# B&R Automation Studio project pneutrunk_plc (part 4)

#### pneutr2_reg_FF_stiff_data.c
```c
/*
 * pneutr2_reg_FF_stiff_data.c
 *
 * Academic License - for use in teaching, academic research, and meeting
 * course requirements at degree granting institutions only.  Not for
 * government, commercial, or other organizational use.
 *
 * Code generation for model "pneutr2_reg_FF_stiff".
 *
 * Model version              : 4.30
 * Simulink Coder version : 9.9 (R2023a) 19-Nov-2022
 * C source code generated on : Thu Feb 15 10:44:02 2024
 *
 * Target selection: bur_grt.tlc
 * Note: GRT includes extra infrastructure and instrumentation for prototyping
 * Embedded hardware selection: Intel->x86/Pentium
 * Code generation objectives: Unspecified
 * Validation result: Not run
 */

#include "pneutr2_reg_FF_stiff.h"

/* Constant parameters (default storage) */
const ConstP_pneutr2_reg_FF_stiff_T pneutr2_reg_FF_stiff_ConstP = {
  /* Expression: coef_1blue_1
   * Referenced by: '<Root>/Constant'
   */
  { 8.5717463150365491E-5, -1.5178110935199764E-6, -5.1507533201889129E-6,
    -4.0104560028142805E-7, -1.7129289185435491E-7, -4.4592625230545557E-7,
    -0.0024294858487422821, 3.9820571035780173E-5, 0.00014194348913824982,
    1.0779763981053751E-5, 4.8691806145412491E-6, 1.2240687126729779E-5,
    0.027186032468499655, -0.000390604161196484, -0.0015838551030587162,
    -0.00011698204244076088, -5.2523210718500108E-5, -0.00013650518202891186,
    -0.15170965057623756, 0.0017650946579940159, 0.0091350333868915647,
    0.00065126150638811556, 0.00027180379442720342, 0.000785516674273971,
    0.43233120736620573, -0.0034156500044472521, -0.028897920231378927,
    -0.0019455068426407257, -0.000689010003804365, -0.0024506052032467382,
    -0.54551465196653193, 0.0011895886985182566, 0.04928011865673651,
    0.002942446648700804, 0.0007337993722779018, 0.0040060166051372123,
    0.50512977080755284, -0.0047809288297403895, -0.03852433507794821,
    -0.0019253109483168883, -0.00010621822149096354, -0.0032474983289435574,
    0.2943360100687234, -0.0340414299034502, 0.038688128292281909,
    0.00078966690125624418, -0.0011243932202755762, 0.0011672777941613569 },

  /* Expression: coef_2green_1
   * Referenced by: '<Root>/Constant1'
   */
  { 3.5806457470463992E-5, 4.2068425285366185E-6, -2.307008943003239E-7,
    -2.8130907926246906E-7, 5.788444538503013E-7, -2.4818480944264519E-7,
    -0.0010926398714506292, -0.00010269300409286399, 5.9242568564171268E-6,
    7.716656677865785E-6, -1.4601073471851697E-5, 7.2919598185173952E-6,
    0.013304512173293481, 0.00098519204569556232, -7.8153808987968122E-5,
    -8.6901728962855031E-5, 0.00014548727107240185, -8.7693471415853716E-5,
    -0.082362007567461509, -0.0047066674356880328, 0.00060563468397506243,
    0.00051035549177713539, -0.00072968678478258365, 0.00055150404791877189,
    0.2700466009571485, 0.01163973248303852, -0.0025271867329235624,
    -0.0016371606003118366, 0.0019364089644989316, -0.0019042555969799237,
    -0.43174345718640667, -0.013838783021252042, 0.0052541678910867822,
    0.0027338218415489421, -0.0025985505984174404, 0.0034092802459716508,
    0.552385933579235, 0.0066940622681189946, -0.013604069710649497,
    -0.0020700479747369879, 0.0015023574386652, -0.0026069405140951157,
    0.031374405216318131, 0.00048138420611595288, -0.035622417341977054,
    0.00018286604488092231, -0.00022698979966827995, 0.0012027861166743492 },

  /* Expression: coef_2green_4
   * Referenced by: '<Root>/Constant10'
   */
  { 3.415320573463566E-7, 9.3053337461778723E-8, -1.1840409221532752E-7,
    -8.3671504125970439E-9, 3.5026579994580658E-9, -2.0473493718581922E-8,
    -2.0177539775413165E-5, -4.5777744650225739E-6, 5.1319620699227294E-6,
    4.6216124370471893E-7, -1.1677319901234268E-7, 9.3377979582771185E-7,
    0.00041167609423549265, 9.3021114154861822E-5, -9.1517441203400879E-5,
    -1.0160859722685084E-5, 1.4151670403326086E-6, -1.7147070588351255E-5,
    -0.0036565061339228488, -0.00098633859891033974, 0.000845215868210654,
    0.00011217230418689672, -6.5999698903405726E-6, 0.00016146662485588915,
    0.012721834814625485, 0.0057771156380495613, -0.0041345518318866188,
    -0.0006595704121746726, -4.6996251846852646E-6, -0.00082145775844466693,
    0.002615152654760115, -0.018645640174938138, 0.010129187197222871,
    0.0020683196398549757, 0.00014406107821792274, 0.0021836634425048385,
    0.20910235409508418, 0.032347602609962139, -0.022366862791594815,
    -0.0034592418366138264, -0.00038747013057998107, -0.0027517673928555875,
    -0.083971676633054743, -0.021473606225994771, -0.045616157291447669,
    0.0022934839006601539, 0.00025030061299072753, 0.0023621895615410903 },

  /* Expression: coef_2green_5
   * Referenced by: '<Root>/Constant11'
   */
  { 1.409263146447497E-6, -6.3007282692451016E-8, 1.1334083156168342E-8,
    9.230072254275008E-9, 2.74393730750942E-9, -4.8715649028139032E-8,
    -6.9391321709493125E-5, 2.0937049836852873E-6, -6.23736765151863E-7,
    -2.3185063573156576E-7, -5.5045992465423964E-8, 2.052665868062509E-6,
    0.0013210734825910666, -2.1292894715980217E-5, 8.565244556977659E-6,
    4.7322333858128524E-7, -1.1535975466056446E-7, -3.453185633002057E-5,
    -0.012145916271257683, 1.5971479419808272E-5, -2.3584719796187389E-5,
    3.192578938792718E-5, 9.9053898987882459E-6, 0.00029591296770094293,
    0.054487936398149417, 0.00099258756801452936, -0.00010064404267846677,
    -0.000347539885728757, -8.7991688376231036E-5, -0.0013616763907182364,
    -0.10407852174157033, -0.0062360441969368831, -0.00016216594324408893,
    0.0014800735016823512, 0.00033604108201676412, 0.0032439882128459277,
    0.3747821795642276, 0.015025591198706953, -0.0083042810415812855,
    -0.0030134939009767536, -0.00064323011865612925, -0.0036482215628668778,
    -0.004527716804257619, -0.010721196323413579, -0.065428003610548333,
    0.0021176098163992788, 0.00057191087607426664, 0.0025894065846387092 },

  /* Pooled Parameter (Expression: coef_2green_6)
   * Referenced by:
   *   '<Root>/Constant12'
   *   '<Root>/Constant18'
   */
  { 1.5081258956513881E-6, -9.046346810421332E-8, 1.4774610225232294E-7,
    -1.7432201593417331E-8, -2.0415701254911555E-9, -5.4201527217183439E-8,
    -7.3850872884215273E-5, 4.5089735689383433E-6, -6.9216959803445692E-6,
    9.8854099646194021E-7, 5.5053432274398986E-8, 2.2269085287207753E-6,
    0.0014042956430304265, -8.8061719814155312E-5, 0.00012698257113709691,
    -2.1915549658526132E-5, 9.0696936183742649E-8, -3.6440744397947455E-5,
    -0.012945155421301551, 0.00086167153240620023, -0.0011917294683145272,
    0.00024280347096503, -1.5415826108399811E-5, 0.00030134255124641181,
    0.058340999413557769, -0.0044888394554316634, 0.0063812751182880829,
    -0.0014299950795206462, 0.00018114458962297672, -0.0013129857525858957,
    -0.1100216315325513, 0.012310894186012916, -0.020155506459850911,
    0.0044334939497109281, -0.00089428426947732876, 0.0028179085747864164,
    0.3631415623276481, -0.01702695159348681, 0.021985457194170679,
    -0.0068753620174089982, 0.0020298400260213797, -0.0023791127843658631,
    0.075563804424678138, 0.010748302896753867, -0.0836195604466876,
    0.0040496210649481768, -0.0015285175321659943, 0.0017237408611272247 },

  /* Expression: coef_3yellow_2
   * Referenced by: '<Root>/Constant13'
   */
  { 6.4204697466336988E-5, -9.4342813666632677E-7, -3.98434162214021E-6,
    -2.4148886551485478E-7, 8.8600986529608742E-8, -3.529598140424027E-7,
    -0.0018407313544118249, 3.0510655304270148E-5, 0.00011104653151774753,
    6.5304832782381205E-6, -2.3344707108276623E-6, 9.65189940926156E-6,
    0.02097491538357809, -0.000387051166283223, -0.0012516712095343016,
    -7.179814137945989E-5, 2.3929248384559622E-5, -0.00010623259914238595,
    -0.12040940291919788, 0.0024820271108887929, 0.0072572354123937189,
    0.00040935377395097877, -0.00011913321761664191, 0.00059895110912360915,
    0.35915882237005048, -0.00861416236255178, -0.022717316237366777,
    -0.0012669750174637902, 0.00029353210289014188, -0.0018144810086714097,
    -0.49859157313593883, 0.015389607153086968, 0.036324219531468319,
    0.0020005131476629814, -0.0003405260446271574, 0.0028020994854614529,
    0.54244105552147959, -0.0045093597732031561, -0.020952154469339943,
    -0.0013450196814645764, 0.00026257246310186223, -0.0019162105937383018,
    0.29795717865338078, 0.029061424095047042, 0.019318582185105713,
    0.00054717765450625067, 0.00043700242127395092, 0.00039781477781437066 },

  /* Expression: coef_3yellow_3
   * Referenced by: '<Root>/Constant14'
   */
  { 6.48259537993542E-8, -1.7774373759257409E-7, -7.808320155327938E-8,
    3.8287288945787542E-8, 5.5727806872203979E-8, -1.8725128684800113E-8,
    -4.45539021636487E-6, 7.0819017739852445E-6, 3.6184317358179945E-6,
    -1.491338534879082E-6, -2.5306282351536662E-6, 8.3322003698335979E-7,
    0.0001039787062549207, -0.00011035727260183309, -6.5873046934394221E-5,
    2.2048281812537434E-5, 4.55402340551219E-5, -1.5071031926050898E-5,
    -0.00098793769743092826, 0.0008614769663412399, 0.00060282012366024156,
    -0.00015092450729609631, -0.00041124074118570862, 0.00014117705330117704,
    0.0022439189860935078, -0.0036459718424953552, -0.0030283199162596912,
    0.00044146382598600064, 0.001946472495698699, -0.00072655371363900109,
    0.018638716969889575, 0.0083590464791400559, 0.0087513807479669085,
    -0.00015550941198203396, -0.0045870757397633247, 0.0020466684533415095,
    0.22372555046354425, 0.00063339384125198669, -0.010561842394564404,
    -0.001534857218792919, 0.0046426063227622064, -0.0031765426227927333,
    0.21321109612687739, 0.062318293620291086, 0.0451142945040786,
    0.0030086997391691591, 0.00020377818613637877, 0.0025250451699678524 },

  /* Expression: coef_3yellow_4
   * Referenced by: '<Root>/Constant15'
   */
  { 8.4131274265651666E-7, -7.4383219245925427E-8, -5.0287276560707072E-8,
    -2.0897845930538842E-8, -6.440085347537078E-9, 6.7481576007548743E-9,
    -4.2672455469044818E-5, 3.6283879790767505E-6, 2.8112580779664218E-6,
    9.4244307790774187E-7, 2.6901736849564227E-7, -2.296605990918742E-7,
    0.00083384358830594434, -6.9445411150021455E-5, -6.1240713144957153E-5,
    -1.7101444974435402E-5, -4.68490716660205E-6, 2.4193458171436571E-6,
    -0.00788467495118846, 0.00068930832276782985, 0.00065222611182779952,
    0.00015873569725615672, 4.6358378535902844E-5, -3.9658563609790317E-6,
    0.036537996817296539, -0.0039525518156003957, -0.0035621008736274875,
    -0.00078838867524841155, -0.0002851236452644136, -7.7595562303436593E-5,
    -0.070575188397405814, 0.012900982665758679, 0.0095640189548843787,
    0.0019881300953568169, 0.00099789757947358433, 0.00046656416534456252,
    0.3319418764249159, -0.010770196313336063, -0.0068139124877474953,
    -0.00213591405094567, -0.0015711778102288714, -0.0010125823263019273,
    0.26470337626557044, 0.065505944077199382, 0.031533925665624365,
    0.001201870952790938, 0.0020343079283254343, 0.00067207527454310662 },

  /* Expression: coef_3yellow_5
   * Referenced by: '<Root>/Constant16'
   */
  { 4.3662861036156025E-7, -5.784570129601148E-8, -1.8954135521594264E-7,
    -2.9674630962163559E-8, -2.3670158106628276E-8, -3.2729331941789806E-8,
    -2.3468166758837827E-5, 2.9856098467640548E-6, 9.3274443686339938E-6,
    1.2416417586297135E-6, 1.0105337017629663E-6, 1.5930389626810239E-6,
    0.0004660426872708893, -5.9127373525058836E-5, -0.00018379559568066587,
    -2.0763013529999418E-5, -1.7410879947845679E-5, -3.1187674050112185E-5,
    -0.0042055718115715946, 0.0006021204215072598, 0.0018509393766251935,
    0.00017594929709408504, 0.00015699137563663005, 0.00031213948479798194,
    0.015724711279660523, -0.0035726500993450289, -0.010165407106281939,
    -0.00078637021515011094, -0.00079166153492090047, -0.0016877500512435754,
    -0.0031156400543770921, 0.012395275356981872, 0.03014616543782124,
    0.0017249015058315486, 0.0021249122383009637, 0.0048258045615070036,
    0.22855436095704232, -0.011417770775931514, -0.039411725580443112,
    -0.0015002089958637552, -0.0023685498365021143, -0.0067663176540085209,
    0.28443427763676743, 0.06817053065209118, 0.057303755590417269,
    0.00074557847875426442, 0.0015466619948328617, 0.0037370891761739767 },

  /* Pooled Parameter (Expression: coef_3yellow_6)
   * Referenced by:
   *   '<Root>/Constant17'
   *   '<Root>/Constant19'
   */
  { 1.7389770421382259E-7, -1.7123638330675637E-7, 9.4499008594265859E-9,
    -5.8708588254654721E-9, -1.3479636927518809E-8, 1.560833585093198E-8,
    -1.1613203471286715E-5, 7.8485997330218131E-6, -1.8241532670320972E-7,
    2.2760816703106266E-7, 5.8832724068270185E-7, -5.7235701233199513E-7,
    0.00025046620896259969, -0.00014165928223837477, -1.93706802370803E-6,
    -3.4949293652347182E-6, -1.0300799281854625E-5, 7.8561723696521691E-6,
    -0.0021106560370579876, 0.0012983291921285149, 7.7781028914489014E-5,
    2.5853236527452207E-5, 9.4488589737110743E-5, -5.0391824164111841E-5,
    0.0035743101337130496, -0.006592046515503186, -0.00080498016859862091,
    -8.37311235355968E-5, -0.00048836064024517238, 0.00015444150339184268,
    0.03814160916752124, 0.018900437397486893, 0.0035312751928995006,
    2.7554344287298178E-5, 0.0013367569729240908, -0.00018514096881816407,
    0.17590112362044411, -0.019836935623231196, 7.6774952652231563E-5,
    0.00037300584604261334, -0.0013435615391459369, -0.00026066130614518947,
    0.46142392823536982, 0.074375754081332887, 0.033324996323250963,
    0.00016012182009621283, 0.00073520569676405992, 0.000681983975687945 },

  /* Expression: coef_1blue_2
   * Referenced by: '<Root>/Constant2'
   */
  { 6.8805425194597416E-5, -5.0957061414343622E-7, -1.5457972525178307E-6,
    -6.6804495762748526E-8, -2.0326730942916425E-7, -1.592771535733192E-7,
    -0.0020076861328312038, 1.2387418133565041E-5, 4.7536114343547258E-5,
    2.2445423401196071E-6, 5.3830284910181655E-6, 4.7423994346354043E-6,
    0.02326778347336618, -0.00011259694455234723, -0.00059908930676579855,
    -3.1187278206521973E-5, -5.6178208735903247E-5, -5.7796033031635973E-5,
    -0.13550439709269863, 0.00042254578575037538, 0.00390965054411615,
    0.00022218858743703064, 0.00028878461318838824, 0.00036313566012097692,
    0.40845960649186464, -0.0001596690481901949, -0.01389459097674536,
    -0.00084049940375010115, -0.00074495341302769573, -0.0012253524173122684,
    -0.56995278689662154, -0.0022970617282296333, 0.025828190334463045,
    0.0015873608396619727, 0.00088390209563778794, 0.0021145632884834453,
    0.59665787978083573, -0.0045164285975585854, -0.017859280842037327,
    -0.0012951931858273045, -0.00044482664081413965, -0.0016581553442656411,
    0.2493667319122021, -0.026109207553320291, 0.021345397673465973,
    0.00056993931435987894, -0.00039599230351878548, 0.0004117320816559158 },

  /* Pooled Parameter (Expression: coef_1blue_6)
   * Referenced by:
   *   '<Root>/Constant20'
   *   '<Root>/Constant7'
   */
  { -8.482401387656442E-8, 1.8922024721926781E-7, -3.8653051637986312E-7,
    -3.2678174480928055E-8, 1.880447821871172E-8, -1.2822794224456168E-8,
    1.6915350706929962E-6, -8.46520419581844E-6, 1.8260895063388544E-5,
    1.3352364435572059E-6, -6.598652293520523E-7, 8.1769478747815578E-7,
    -6.4520565065795527E-6, 0.00014750653726755962, -0.0003476823679280495,
    -2.1618373462681182E-5, 7.8376482422089821E-6, -1.9857256883187996E-5,
    0.00017248832659086518, -0.0012863621148176438, 0.0034326081784590411,
    0.0001764797024344746, -2.8647563822075195E-5, 0.00023871706739248702,
    -0.00509888879868316, 0.0061192208764403047, -0.018906833199680808,
    -0.0007655906488482256, -0.00011253868356740794, -0.0015280157931335438,
    0.042005527755441183, -0.016229623272152709, 0.05797438180721573,
    0.0017206754753116634, 0.0011750481477870076, 0.00518174219812922,
    0.25162359279096436, 0.012815884510758872, -0.085082859600351474,
    -0.0020876564441693131, -0.0033018769498668692, -0.0087796216724272923,
    0.088402040598522608, -0.064192606835404453, 0.087578799157964016,
    0.0020707162045730033, 0.0018421383794582453, 0.0055748188793970505 },

  /* Expression: coef_3yellow_1
   * Referenced by: '<Root>/Constant3'
   */
  { 7.0192131586256317E-5, 1.2977198686205759E-6, -5.5571290250705513E-6,
    -4.79340188517608E-7, -9.4819440719696464E-8, -4.284483956134012E-7,
    -0.0019777629168876536, -3.1672961282187759E-5, 0.00015371415729669983,
    1.2304544272507984E-5, 2.2231831201926792E-6, 1.1908428533383876E-5,
    0.02198870564343576, 0.00029899890562501066, -0.001721213425076836,
    -0.00012613116841534447, -2.0663195033571994E-5, -0.00013483353433428347,
    -0.12173838504903266, -0.0013453385352150168, 0.0099688064773889914,
    0.00065690233120104728, 0.00010100455976903478, 0.00078899402332532171,
    0.34334397402467365, 0.00272896932065054, -0.031593480309384775,
    -0.0018205946834633174, -0.00028992744729897736, -0.0025034134427869659,
    -0.4273116869060552, -0.0013021586849929355, 0.052918295813197326,
    0.0025379227628717174, 0.00049392618790492567, 0.0041456352312311262,
    0.4271806989365543, 0.0047301397271836809, -0.037856026736010559,
    -0.0015320371928851516, -0.00037071463595379073, -0.0033021318563182028,
    0.30066005013967406, 0.033716002450655279, 0.033067942069331432,
    0.000755329711910434, 0.00087321497388740158, 0.0011326660929602316 },

  /* Expression: coef_1blue_3
   * Referenced by: '<Root>/Constant4'
   */
  { -6.87039592092718E-7, 2.7397086829932237E-7, -3.2684627499899603E-7,
    -4.6654219126960229E-8, -1.7025805182385262E-8, -7.1035135706855437E-9,
    2.491824277460112E-5, -1.0993006031749188E-5, 1.4945724368839632E-5,
    1.9598316440108521E-6, 8.6187422580204285E-7, 4.9619648608464926E-7,
    -0.00037451180905163738, 0.00017366919763100707, -0.00027648100689608404,
    -3.2844279876213038E-5, -1.697373374485846E-5, -1.2700924253991477E-5,
    0.0034675352360980429, -0.0013723548375873726, 0.0026572919564385512,
    0.00027833828005838088, 0.000164929704244049, 0.000156516149348449,
    -0.024396844251214307, 0.0057531176572915331, -0.014237435617272897,
    -0.00124884077318305, -0.000825643341125968, -0.0010058083347592546,
    0.11412199121860407, -0.012337656381244136, 0.042444713486128174,
    0.002846531771851347, 0.0020211766310428867, 0.003392567101489787,
    0.13841237933708728, 0.0013799439664535747, -0.061479686753332707,
    -0.0030605232152760226, -0.0021269181943356619, -0.0058577489821760829,
    0.4218191857644718, -0.0680306271879334, 0.082616432288031991,
    0.0018661063635620929, -0.00078014099479087556, 0.0043230499199038 },

  /* Expression: coef_1blue_4
   * Referenced by: '<Root>/Constant5'
   */
  { -3.1072883946418533E-7, 3.9051524168297835E-8, -4.4738920574513E-8,
    -1.4261453975904657E-8, -2.4524445372588755E-8, -8.6581555252886952E-9,
    1.1832112622050945E-5, -1.8478700295428403E-6, 2.8157736675211269E-6,
    6.4348105019410092E-7, 1.0715173793584769E-6, 4.4428009382398351E-7,
    -0.00019640741291831733, 3.5493301079018969E-5, -6.8318351008526951E-5,
    -1.1877259782247793E-5, -1.8565837129361158E-5, -9.18999874018573E-6,
    0.0021613548617786865, -0.00035580706199814439, 0.00082431655018391792,
    0.00011352525979972025, 0.00016052432147366659, 9.6237365088613279E-5,
    -0.018244224281010604, 0.0020150599383139249, -0.0053371562668590011,
    -0.00058967044793498168, -0.00071771672797585307, -0.000536262564353319,
    0.0951514815538755, -0.0057446224427062089, 0.018400819504468206,
    0.0016094394547771715, 0.0016038214220086954, 0.0015689643049010451,
    0.18792703443323883, -0.0044841352892458957, -0.026866914625506944,
    -0.0022463580064703793, -0.0017678331505959213, -0.0024549929470950782,
    0.51635423944282277, -0.058817475277171759, 0.05801974580408828,
    0.0019722167842653351, -0.00031518055683877043, 0.0017747966459091143 },

  /* Expression: coef_1blue_5
   * Referenced by: '<Root>/Constant6'
   */
  { -1.2764738249740704E-6, 4.026116322326337E-7, -3.681597343130841E-7,
    -3.8884837885108559E-8, 5.6507820756228694E-8, -1.6515995353244439E-9,
    5.4349278962288705E-5, -1.6969515485371073E-5, 1.6455802774321442E-5,
    1.6728556957522296E-6, -2.4511588355149069E-6, 1.734257128706172E-7,
    -0.00093049449542566016, 0.00028238016678062982, -0.00029562274019560007,
    -2.9001430808122702E-5, 4.2774077657753696E-5, -5.5075353062715733E-6,
    0.00841399437399872, -0.0023713258687265756, 0.0027439345780921427,
    0.00025907510422729834, -0.00038656026559018373, 7.8075333200169645E-5,
    -0.04508116549745423, 0.01074102507190572, -0.014136276966891358,
    -0.0012644680315192763, 0.0019328812927384934, -0.00055799863995609385,
    0.14748385419878324, -0.025800305766340927, 0.04027223983768715,
    0.0033007799186923212, -0.005224841084560102, 0.0020683496469081335,
    0.12301952312650957, 0.019299343268092715, -0.053556575170859905,
    -0.0043627775154514679, 0.006707713841550964, -0.0039199792773620288,
    0.37788579430972047, -0.0714827213544873, 0.07061563482482891,
    0.0032675749283996589, -0.0041427994547245375, 0.0030285163329780468 },

  /* Expression: coef_2green_2
   * Referenced by: '<Root>/Constant8'
   */
  { 6.2701038492250791E-5, -6.0760977071365537E-8, 1.6275461434525351E-8,
    -1.7119151076355381E-7, -4.5405928686195757E-8, -2.2571974234984949E-7,
    -0.0017462827997451363, 1.5683895488068119E-6, -2.6737148103855792E-6,
    4.8441669785717E-6, 9.43146866783444E-7, 5.9997793789077907E-6,
    0.019291115446101428, -1.7052537276564115E-5, 4.7218096294053983E-5,
    -5.5503600229903927E-5, -6.5788412283737411E-6, -6.4855595417819692E-5,
    -0.10747683267287286, 0.0001098714132076877, -0.00033469851695099235,
    0.00032625511060371262, 1.373717016903375E-5, 0.00036591705625992028,
    0.31398448594826944, -0.00044246330373362086, 0.001244093281090631,
    -0.0010311061532886925, 3.4013866624391472E-5, -0.0011423700773628754,
    -0.43549488523258423, 0.0009533232107337557, -0.0023792310895955461,
    0.0016849908072488762, -0.00018564290581707784, 0.0018930398793588676,
    0.48201224871436416, -0.00031072981032643669, -0.007469539551164495,
    -0.0012952847385186157, 0.00025357114323703661, -0.0014449349202602733,
    0.026146653561975309, -0.0001194944631572856, -0.023737088442451627,
    0.0002070876837847607, -0.00021331332931719214, 0.000858086587181055 },

  /* Expression: coef_2green_3
   * Referenced by: '<Root>/Constant9'
   */
  { 8.0095503939967249E-7, 1.3128794965903748E-7, 4.1778899945657014E-8,
    -2.693826482723759E-8, -2.3144078388512325E-8, -2.3058705434125125E-8,
    -4.0332713634069196E-5, -5.9336765963705979E-6, -1.2775678337040855E-6,
    1.2209213699823443E-6, 1.0250350318183633E-6, 1.0259563007213323E-6,
    0.0007776626160830068, 0.00010828256376351291, 8.98254387057521E-6,
    -2.2111726220952415E-5, -1.8391394625940988E-5, -1.8458087652190355E-5,
    -0.0071807745521049494, -0.0010116709542780026, 6.2074231318600534E-5,
    0.00020149896288088105, 0.00017117948656953191, 0.00017173362969902708,
    0.032142271011353626, 0.0050710137886939609, -0.00089484121984427728,
    -0.00096010831844634882, -0.00087972202926074551, -0.00087426019145385025,
    -0.060012439301404222, -0.013216308890823782, 0.00261001379548545,
    0.0022906342038700117, 0.0024474821943361656, 0.0023511722291509529,
    0.33673447258924616, 0.01727966657744439, -0.010081101210561542,
    -0.0025754435708828442, -0.0032985861784250053, -0.002917863803891091,
    0.034792323564463948, -0.00552555850616554, -0.070027601305080039,
    0.00078499732670345482, 0.0014126253416459848, 0.0018419585865831554 },

  /* Expression: (hodnoty(:,1))
   * Referenced by: '<S36>/z2pressure'
   */
  { 118.39, 138.5, 145.8, 148.48, 150.88, 151.44, 152.75 },

  /* Computed Parameter: z2pressure_tableData
   * Referenced by: '<S36>/z2pressure'
   */
  { 0.0F, 1.0F, 2.0F, 3.0F, 4.0F, 5.0F, 6.0F }
};
```

#### rtGetInf.c
```c
/*
 * rtGetInf.c
 *
 * Academic License - for use in teaching, academic research, and meeting
 * course requirements at degree granting institutions only.  Not for
 * government, commercial, or other organizational use.
 *
 * Code generation for model "pneutr2_reg_FF_stiff".
 *
 * Model version              : 4.30
 * Simulink Coder version : 9.9 (R2023a) 19-Nov-2022
 * C source code generated on : Thu Feb 15 10:44:02 2024
 *
 * Target selection: bur_grt.tlc
 * Note: GRT includes extra infrastructure and instrumentation for prototyping
 * Embedded hardware selection: Intel->x86/Pentium
 * Code generation objectives: Unspecified
 * Validation result: Not run
 */

#include "rtwtypes.h"
#include "rtGetInf.h"
#include <stddef.h>
#include "rt_nonfinite.h"
#define NumBitsPerChar                 8U

/*
 * Initialize rtInf needed by the generated code.
 * Inf is initialized as non-signaling. Assumes IEEE.
 */
real_T rtGetInf(void)
{
  size_t bitsPerReal = sizeof(real_T) * (NumBitsPerChar);
  real_T inf = 0.0;
  if (bitsPerReal == 32U) {
    inf = rtGetInfF();
  } else {
    uint16_T one = 1U;
    enum {
      LittleEndian,
      BigEndian
    } machByteOrder = (*((uint8_T *) &one) == 1U) ? LittleEndian : BigEndian;
    switch (machByteOrder) {
     case LittleEndian:
      {
        union {
          LittleEndianIEEEDouble bitVal;
          real_T fltVal;
        } tmpVal;

        tmpVal.bitVal.words.wordH = 0x7FF00000U;
        tmpVal.bitVal.words.wordL = 0x00000000U;
        inf = tmpVal.fltVal;
        break;
      }

     case BigEndian:
      {
        union {
          BigEndianIEEEDouble bitVal;
          real_T fltVal;
        } tmpVal;

        tmpVal.bitVal.words.wordH = 0x7FF00000U;
        tmpVal.bitVal.words.wordL = 0x00000000U;
        inf = tmpVal.fltVal;
        break;
      }
    }
  }

  return inf;
}

/*
 * Initialize rtInfF needed by the generated code.
 * Inf is initialized as non-signaling. Assumes IEEE.
 */
real32_T rtGetInfF(void)
{
  IEEESingle infF;
  infF.wordL.wordLuint = 0x7F800000U;
  return infF.wordL.wordLreal;
}

/*
 * Initialize rtMinusInf needed by the generated code.
 * Inf is initialized as non-signaling. Assumes IEEE.
 */
real_T rtGetMinusInf(void)
{
  size_t bitsPerReal = sizeof(real_T) * (NumBitsPerChar);
  real_T minf = 0.0;
  if (bitsPerReal == 32U) {
    minf = rtGetMinusInfF();
  } else {
    uint16_T one = 1U;
    enum {
      LittleEndian,
      BigEndian
    } machByteOrder = (*((uint8_T *) &one) == 1U) ? LittleEndian : BigEndian;
    switch (machByteOrder) {
     case LittleEndian:
      {
        union {
          LittleEndianIEEEDouble bitVal;
          real_T fltVal;
        } tmpVal;

        tmpVal.bitVal.words.wordH = 0xFFF00000U;
        tmpVal.bitVal.words.wordL = 0x00000000U;
        minf = tmpVal.fltVal;
        break;
      }

     case BigEndian:
      {
        union {
          BigEndianIEEEDouble bitVal;
          real_T fltVal;
        } tmpVal;

        tmpVal.bitVal.words.wordH = 0xFFF00000U;
        tmpVal.bitVal.words.wordL = 0x00000000U;
        minf = tmpVal.fltVal;
        break;
      }
    }
  }

  return minf;
}

/*
 * Initialize rtMinusInfF needed by the generated code.
 * Inf is initialized as non-signaling. Assumes IEEE.
 */
real32_T rtGetMinusInfF(void)
{
  IEEESingle minfF;
  minfF.wordL.wordLuint = 0xFF800000U;
  return minfF.wordL.wordLreal;
}
```

#### solo_reg.c
```c
/********************************************************************
 * COPYRIGHT -- B&R Industrial Automation GmbH
 ********************************************************************
 * Program: solo_reg
 * File: solo_reg.c
 * Author: varga
 * Last modified by: varga
 * Created: 15-Feb-2024 10:44:14
 * Last modified: Thu Feb 15 10:41:29 2024
 * Model Version: 4.30
 * Description:
 * modified Comment:
 ********************************************************************
 * Implementation of program solo_reg
 ********************************************************************
 * Generated with B&R Automation Studio Target for Simulink V6.8
 * (GRT based)
 ********************************************************************/

#define _ASMATH_
#define ASMATH_
#define _ASMATH_H
#define ASMATH_H
#define _ASMATH_H_
#define ASMATH_H_
#define _ASSTRING_
#define ASSTRING_
#define _ASSTRING_H
#define ASSTRING_H
#define _ASSTRING_H_
#define ASSTRING_H_

#include <bur/plctypes.h>

#ifdef _DEFAULT_INCLUDES
 #include <AsDefault.h>
#endif

#include "rtwtypes.h"
#include "rtmodel.h"

#define EXPAND_CONCAT(name1,name2) name1 ## name2
#define CONCAT(name1,name2) EXPAND_CONCAT(name1,name2)
#define RT_MODEL            CONCAT(MODEL,_rtModel)

#ifdef __cplusplus

extern "C" {

#endif

extern RT_MODEL *MODEL(void);

extern void MdlInitializeSizes(void);
extern void MdlInitializeSampleTimes(void);
extern void MdlStart(void);
extern void MdlOutputs(int_T tid);
extern void MdlUpdate(int_T tid);
extern void MdlTerminate(void);

#ifdef __cplusplus

}

#endif

#ifdef __cplusplus
    unsigned long bur_heap_size = 6553500;
#endif

void _INIT mainINIT( void )
{

    UDINT st_ident;
    RTInfo_typ rt_info;
    rt_info.enable = 1;
    RTInfo(&rt_info);
    if (rt_info.cycle_time != 16000)
    {
      /* cycle time does not match Simulink fixed-step size */
      ST_ident("solo_reg", 0, &st_ident);
      ST_tmp_suspend(st_ident);
      ERR_warning(33310, 0);
    }

	RT_MODEL  *S;

	S = MODEL();

	MdlInitializeSizes();
	MdlInitializeSampleTimes();
	MdlStart();

}

void _CYCLIC mainCYCLIC( void )
{
	MdlOutputs(0);
	MdlUpdate(0);

}

void _EXIT mainEXIT( void )
{
	MdlTerminate();

}

/*****************************************************************************
  Task sample time: 0.016s
 *****************************************************************************/

/*****************************************************************************
   B&R Automation Studio Target for Simulink Version: V6.8.0 (22-Mar-2023)
 *****************************************************************************/
```

### Program Logical/test_input (ANSIC, version 1.00.0)

#### rtGetInf.c
```c
/*
 * rtGetInf.c
 *
 * Academic License - for use in teaching, academic research, and meeting
 * course requirements at degree granting institutions only.  Not for
 * government, commercial, or other organizational use.
 *
 * Code generation for model "simulink_2_plc".
 *
 * Model version              : 1.4
 * Simulink Coder version : 9.9 (R2023a) 19-Nov-2022
 * C source code generated on : Tue Feb  6 09:08:04 2024
 *
 * Target selection: bur_grt.tlc
 * Note: GRT includes extra infrastructure and instrumentation for prototyping
 * Embedded hardware selection: Intel->x86/Pentium
 * Code generation objectives: Unspecified
 * Validation result: Not run
 */

#include "rtwtypes.h"
#include "rtGetInf.h"
#include <stddef.h>
#include "rt_nonfinite.h"
#define NumBitsPerChar                 8U

/*
 * Initialize rtInf needed by the generated code.
 * Inf is initialized as non-signaling. Assumes IEEE.
 */
real_T rtGetInf(void)
{
  size_t bitsPerReal = sizeof(real_T) * (NumBitsPerChar);
  real_T inf = 0.0;
  if (bitsPerReal == 32U) {
    inf = rtGetInfF();
  } else {
    uint16_T one = 1U;
    enum {
      LittleEndian,
      BigEndian
    } machByteOrder = (*((uint8_T *) &one) == 1U) ? LittleEndian : BigEndian;
    switch (machByteOrder) {
     case LittleEndian:
      {
        union {
          LittleEndianIEEEDouble bitVal;
          real_T fltVal;
        } tmpVal;

        tmpVal.bitVal.words.wordH = 0x7FF00000U;
        tmpVal.bitVal.words.wordL = 0x00000000U;
        inf = tmpVal.fltVal;
        break;
      }

     case BigEndian:
      {
        union {
          BigEndianIEEEDouble bitVal;
          real_T fltVal;
        } tmpVal;

        tmpVal.bitVal.words.wordH = 0x7FF00000U;
        tmpVal.bitVal.words.wordL = 0x00000000U;
        inf = tmpVal.fltVal;
        break;
      }
    }
  }

  return inf;
}

/*
 * Initialize rtInfF needed by the generated code.
 * Inf is initialized as non-signaling. Assumes IEEE.
 */
real32_T rtGetInfF(void)
{
  IEEESingle infF;
  infF.wordL.wordLuint = 0x7F800000U;
  return infF.wordL.wordLreal;
}

/*
 * Initialize rtMinusInf needed by the generated code.
 * Inf is initialized as non-signaling. Assumes IEEE.
 */
real_T rtGetMinusInf(void)
{
  size_t bitsPerReal = sizeof(real_T) * (NumBitsPerChar);
  real_T minf = 0.0;
  if (bitsPerReal == 32U) {
    minf = rtGetMinusInfF();
  } else {
    uint16_T one = 1U;
    enum {
      LittleEndian,
      BigEndian
    } machByteOrder = (*((uint8_T *) &one) == 1U) ? LittleEndian : BigEndian;
    switch (machByteOrder) {
     case LittleEndian:
      {
        union {
          LittleEndianIEEEDouble bitVal;
          real_T fltVal;
        } tmpVal;

        tmpVal.bitVal.words.wordH = 0xFFF00000U;
        tmpVal.bitVal.words.wordL = 0x00000000U;
        minf = tmpVal.fltVal;
        break;
      }

     case BigEndian:
      {
        union {
          BigEndianIEEEDouble bitVal;
          real_T fltVal;
        } tmpVal;

        tmpVal.bitVal.words.wordH = 0xFFF00000U;
        tmpVal.bitVal.words.wordL = 0x00000000U;
        minf = tmpVal.fltVal;
        break;
      }
    }
  }

  return minf;
}

/*
 * Initialize rtMinusInfF needed by the generated code.
 * Inf is initialized as non-signaling. Assumes IEEE.
 */
real32_T rtGetMinusInfF(void)
{
  IEEESingle minfF;
  minfF.wordL.wordLuint = 0xFF800000U;
  return minfF.wordL.wordLreal;
}
```

#### rtwtypes.h
```c
/*
 * rtwtypes.h
 *
 * Academic License - for use in teaching, academic research, and meeting
 * course requirements at degree granting institutions only.  Not for
 * government, commercial, or other organizational use.
 *
 * Code generation for model "simulink_2_plc".
 *
 * Model version              : 1.4
 * Simulink Coder version : 9.9 (R2023a) 19-Nov-2022
 * C source code generated on : Tue Feb  6 09:08:04 2024
 *
 * Target selection: bur_grt.tlc
 * Note: GRT includes extra infrastructure and instrumentation for prototyping
 * Embedded hardware selection: Intel->x86/Pentium
 * Code generation objectives: Unspecified
 * Validation result: Not run
 */

#ifndef RTWTYPES_H
#define RTWTYPES_H
#include "tmwtypes.h"
#ifndef POINTER_T
#define POINTER_T

typedef void * pointer_T;

#endif

/* Logical type definitions */
#if (!defined(__cplusplus))
#ifndef false
#define false                          (0U)
#endif

#ifndef true
#define true                           (1U)
#endif
#endif
#endif                                 /* RTWTYPES_H */
```

#### simulink_2_plc_data.c
```c
/*
 * simulink_2_plc_data.c
 *
 * Academic License - for use in teaching, academic research, and meeting
 * course requirements at degree granting institutions only.  Not for
 * government, commercial, or other organizational use.
 *
 * Code generation for model "simulink_2_plc".
 *
 * Model version              : 1.4
 * Simulink Coder version : 9.9 (R2023a) 19-Nov-2022
 * C source code generated on : Tue Feb  6 09:08:04 2024
 *
 * Target selection: bur_grt.tlc
 * Note: GRT includes extra infrastructure and instrumentation for prototyping
 * Embedded hardware selection: Intel->x86/Pentium
 * Code generation objectives: Unspecified
 * Validation result: Not run
 */

#include "simulink_2_plc.h"

/* Block parameters (default storage) */
P_simulink_2_plc_T simulink_2_plc_P = {
  /* Expression: 8
   * Referenced by: '<Root>/Sine Wave'
   */
  8.0,

  /* Expression: 0
   * Referenced by: '<Root>/Sine Wave'
   */
  0.0,

  /* Expression: 1.4
   * Referenced by: '<Root>/Sine Wave'
   */
  1.4,

  /* Expression: 0
   * Referenced by: '<Root>/Sine Wave'
   */
  0.0,

  /* Expression: 6
   * Referenced by: '<Root>/Sine Wave1'
   */
  6.0,

  /* Expression: 0
   * Referenced by: '<Root>/Sine Wave1'
   */
  0.0,

  /* Expression: 0.5
   * Referenced by: '<Root>/Sine Wave1'
   */
  0.5,

  /* Expression: 0
   * Referenced by: '<Root>/Sine Wave1'
   */
  0.0,

  /* Computed Parameter: Gain_Gain
   * Referenced by: '<Root>/Gain'
   */
  1.0F,

  /* Computed Parameter: Gain1_Gain
   * Referenced by: '<Root>/Gain1'
   */
  1.0F
};
```

#### simulink_2_plc_private.h
```c
/*
 * simulink_2_plc_private.h
 *
 * Academic License - for use in teaching, academic research, and meeting
 * course requirements at degree granting institutions only.  Not for
 * government, commercial, or other organizational use.
 *
 * Code generation for model "simulink_2_plc".
 *
 * Model version              : 1.4
 * Simulink Coder version : 9.9 (R2023a) 19-Nov-2022
 * C source code generated on : Tue Feb  6 09:08:04 2024
 *
 * Target selection: bur_grt.tlc
 * Note: GRT includes extra infrastructure and instrumentation for prototyping
 * Embedded hardware selection: Intel->x86/Pentium
 * Code generation objectives: Unspecified
 * Validation result: Not run
 */

#ifndef RTW_HEADER_simulink_2_plc_private_h_
#define RTW_HEADER_simulink_2_plc_private_h_
#include "rtwtypes.h"
#include "multiword_types.h"
#include "zero_crossing_types.h"
#include "simulink_2_plc_types.h"
#endif                                /* RTW_HEADER_simulink_2_plc_private_h_ */
```

Listed in the project but not available here: Logical/Source/UDP/LibAsUDP1_ST.typ, Logical/Source/UDP/LibAsUDP1_ST.var, Logical/Source/UDP/Server, Logical/Source/UDP/Client/Client.var, Logical/Source/MATLAB_includes, Logical/Source/riadenie.var, Logical/Source/Identifikacia, Logical/meranie/local.typ, Logical/meranie/local.var, Logical/meranie/meranie.c, Logical/meranie/pneutrunkMeranie.h, Logical/meranie/pneutrunkMeranie_dt.h, Logical/meranie/pneutrunkMeranie_private.h, Logical/meranie/pneutrunkMeranie_types.h, Logical/meranie/rtGetInf.c, Logical/meranie/rtGetInf.h, Logical/meranie/rtGetNaN.c, Logical/meranie/rtGetNaN.h, Logical/meranie/rt_defines.h, Logical/meranie/rt_nonfinite.c, Logical/meranie/rt_nonfinite.h, Logical/meranie/rtmodel.h, Logical/meranie/rtwtypes.h, Logical/meranie/zero_crossing_types.h, Logical/meranie/extmode/bur_logging.c, Logical/meranie/extmode/bur_logging.h, Logical/meranie/extmode/ext_svr.c, Logical/meranie/extmode/ext_work.c, Logical/meranie/extmode/mem_mgr.c, Logical/meranie/extmode/rtiostream_interface.c, Logical/meranie/extmode/rtiostream_tcpip_static.c, Logical/meranie/extmode/updown.c, Logical/MATLAB_includes/R2021b/MatlabDataArray.hpp, Logical/MATLAB_includes/R2021b/MatlabEngine.hpp, Logical/MATLAB_includes/R2021b/bio_sig.h, Logical/MATLAB_includes/R2021b/blas.h, Logical/MATLAB_includes/R2021b/blascompat32.h, Logical/MATLAB_includes/R2021b/cg_matrx.h, Logical/MATLAB_includes/R2021b/cg_sfun.h, Logical/MATLAB_includes/R2021b/cgxeooprt.h, Logical/MATLAB_includes/R2021b/cgxert.h, Logical/MATLAB_includes/R2021b/covrt.h, Logical/MATLAB_includes/R2021b/dt_info.h, Logical/MATLAB_includes/R2021b/emlrt.h, Logical/MATLAB_includes/R2021b/engine.h, Logical/MATLAB_includes/R2021b/ext_share.h, Logical/MATLAB_includes/R2021b/ext_svr.h, Logical/MATLAB_includes/R2021b/ext_svr_transport.h, Logical/MATLAB_includes/R2021b/ext_test.h, Logical/MATLAB_includes/R2021b/ext_types.h, Logical/MATLAB_includes/R2021b/ext_work.h, Logical/MATLAB_includes/R2021b/fintrf.h, Logical/MATLAB_includes/R2021b/fixedpoint.h, Logical/MATLAB_includes/R2021b/fixpoint_spec.h, Logical/MATLAB_includes/R2021b/i18n_c_api.h, Logical/MATLAB_includes/R2021b/io64.h, Logical/MATLAB_includes/R2021b/lapack.h, Logical/MATLAB_includes/R2021b/lapacke.h, Logical/MATLAB_includes/R2021b/lapacke_config.h, Logical/MATLAB_includes/R2021b/libmwjpegreader.h, Logical/MATLAB_includes/R2021b/libmwrgb2gray_tbb.h, Logical/MATLAB_includes/R2021b/libmwrgb2hsv_tbb.h, Logical/MATLAB_includes/R2021b/libmwslsa_sim.h, Logical/MATLAB_includes/R2021b/mat.h, Logical/MATLAB_includes/R2021b/matrix.h, Logical/MATLAB_includes/R2021b/mdl_info.h, Logical/MATLAB_includes/R2021b/mem_mgr.h, Logical/MATLAB_includes/R2021b/mex.h, Logical/MATLAB_includes/R2021b/mwmathutil.h, Logical/MATLAB_includes/R2021b/odesup.h, Logical/MATLAB_includes/R2021b/polygonBoolean.h, Logical/MATLAB_includes/R2021b/pt_info.h, Logical/MATLAB_includes/R2021b/rt_logging.h, Logical/MATLAB_includes/R2021b/rt_logging_mmi.h, Logical/MATLAB_includes/R2021b/rt_math.h, Logical/MATLAB_includes/R2021b/rt_matrx.h, Logical/MATLAB_includes/R2021b/rt_mxclassid.h, Logical/MATLAB_includes/R2021b/rt_sim.h, Logical/MATLAB_includes/R2021b/rtiostream.h, Logical/MATLAB_includes/R2021b/rtmcmacros.h, Logical/MATLAB_includes/R2021b/rtmmacros.h, Logical/MATLAB_includes/R2021b/rtsplntypes.h, Logical/MATLAB_includes/R2021b/rtw_capi.h, Logical/MATLAB_includes/R2021b/rtw_capi_examples.h, Logical/MATLAB_includes/R2021b/rtw_continuous.h, Logical/MATLAB_includes/R2021b/rtw_extmode.h, Logical/MATLAB_includes/R2021b/rtw_linux.h, Logical/MATLAB_includes/R2021b/rtw_linux_mac.h, Logical/MATLAB_includes/R2021b/rtw_matlogging.h, Logical/MATLAB_includes/R2021b/rtw_matlogging_simtarget.h, Logical/MATLAB_includes/R2021b/rtw_modelmap.h, Logical/MATLAB_includes/R2021b/rtw_modelmap_logging.h, Logical/MATLAB_includes/R2021b/rtw_msvc_lshift.h, Logical/MATLAB_includes/R2021b/rtw_solver.h, Logical/MATLAB_includes/R2021b/rtw_storage.h, Logical/MATLAB_includes/R2021b/rtw_windows.h, Logical/MATLAB_includes/R2021b/sfcn_bridge.h, Logical/MATLAB_includes/R2021b/sfcn_loader_c_api.h, Logical/MATLAB_includes/R2021b/sfun_rtwcg.hpp, Logical/MATLAB_includes/R2021b/sigmapdef_sfcn.h, Logical/MATLAB_includes/R2021b/sigregdef.h, Logical/MATLAB_includes/R2021b/sigstream_rtw.h, Logical/MATLAB_includes/R2021b/simlogCIntrf.h, Logical/MATLAB_includes/R2021b/simstruc.h, Logical/MATLAB_includes/R2021b/simstruc_64_internal.h, Logical/MATLAB_includes/R2021b/simstruc_compcond.h, Logical/MATLAB_includes/R2021b/simstruc_debug.h, Logical/MATLAB_includes/R2021b/simstruc_def.h, Logical/MATLAB_includes/R2021b/simstruc_implement.h, Logical/MATLAB_includes/R2021b/simstruc_internal.h, Logical/MATLAB_includes/R2021b/simstruc_internal_types.h, Logical/MATLAB_includes/R2021b/simstruc_types.h, Logical/MATLAB_includes/R2021b/simulink.h, Logical/MATLAB_includes/R2021b/simulink2.h, Logical/MATLAB_includes/R2021b/simulink_solver_api.h, Logical/MATLAB_includes/R2021b/slImageTypes.h, Logical/MATLAB_includes/R2021b/sl_common_types_def.h, Logical/MATLAB_includes/R2021b/sl_datatype_access.h, Logical/MATLAB_includes/R2021b/sl_fileio_rtw.h, Logical/MATLAB_includes/R2021b/sl_fixpt.h, Logical/MATLAB_includes/R2021b/sl_prodhwdevicetype.h, Logical/MATLAB_includes/R2021b/sl_report_types.h, Logical/MATLAB_includes/R2021b/sl_sample_time_defs.h, Logical/MATLAB_includes/R2021b/sl_sfcn_st_api.h, Logical/MATLAB_includes/R2021b/sl_solver_rtw.h, Logical/MATLAB_includes/R2021b/sl_types_def.h, Logical/MATLAB_includes/R2021b/slccrt.h, Logical/MATLAB_includes/R2021b/slexec_block_runtime_service.h, Logical/MATLAB_includes/R2021b/slexec_parallel.h, Logical/MATLAB_includes/R2021b/slexec_simbridge.h, Logical/MATLAB_includes/R2021b/slexec_simstruct_bridge.h, Logical/MATLAB_includes/R2021b/slexec_ssExecutionInfo.h, Logical/MATLAB_includes/R2021b/slexec_vm_lookup_functions.h, Logical/MATLAB_includes/R2021b/slexec_vm_rt_functions.h, Logical/MATLAB_includes/R2021b/slexec_vm_simstruct_bridge.h, Logical/MATLAB_includes/R2021b/slexec_vm_zc_functions.h, Logical/MATLAB_includes/R2021b/slsa_sim_engine.h, Logical/MATLAB_includes/R2021b/slsv_diagnostic_codegen_c_api.h, Logical/MATLAB_includes/R2021b/slsv_diagnostic_deployment_c_api.h, Logical/MATLAB_includes/R2021b/slsv_diagnostic_logger_type.h, Logical/MATLAB_includes/R2021b/slsv_mexhelper.h, Logical/MATLAB_includes/R2021b/solver_zc.h, Logical/MATLAB_includes/R2021b/sysran_types.h, Logical/MATLAB_includes/R2021b/tmwtypes.h, Logical/MATLAB_includes/R2021b/updown.h, Logical/MATLAB_includes/R2021b/updown_util.h, Logical/MATLAB_includes/R2021b/upsup_public.h, Logical/MATLAB_includes/R2021b/sf_runtime, Logical/MATLAB_includes/R2023a/sf_runtime/MessageServiceLayer.h, Logical/MATLAB_includes/R2023a/sf_runtime/sf_runtime_errors.h, Logical/MATLAB_includes/R2023a/sf_runtime/sf_runtime_spec.h, Logical/MATLAB_includes/R2023a/sf_runtime/sf_runtime_types.h, Logical/MATLAB_includes/R2023a/sf_runtime/sf_test_language.h, Logical/MATLAB_includes/R2023a/sf_runtime/sfc_api.h, Logical/MATLAB_includes/R2023a/sf_runtime/sfc_messages.h, Logical/MATLAB_includes/R2023a/sf_runtime/sfc_mex.h, Logical/MATLAB_includes/R2023a/sf_runtime/sfc_sdi.h, Logical/MATLAB_includes/R2023a/sf_runtime/sfc_sf.h, Logical/MATLAB_includes/R2023a/sf_runtime/sfcdebug.h, Logical/MATLAB_includes/R2023a/sf_runtime/slTestResult.h, Logical/MATLAB_includes/R2023a/sf_runtime/slTestTypes.h, Logical/MATLAB_includes/R2023a/sf_runtime/utils.h, Logical/MATLAB_includes/R2023a/sf_runtime/ChartInfoStruct.h, Logical/MATLAB_includes/R2023a/sf_runtime/DebuggerRuntimeInterface.h, Logical/MATLAB_includes/R2023a/sf_runtime/sf_partitioning_execution_bridge.h, Logical/test_input/local.typ, Logical/test_input/local.var, Logical/test_input/multiword_types.h, Logical/test_input/rtGetInf.h, Logical/test_input/rtGetNaN.c, Logical/test_input/rtGetNaN.h, Logical/test_input/rt_defines.h, Logical/test_input/rt_nonfinite.c, Logical/test_input/rt_nonfinite.h, Logical/test_input/rtmodel.h, Logical/test_input/simulink_2_plc.c, Logical/test_input/simulink_2_plc.h, Logical/test_input/simulink_2_plc_dt.h, Logical/test_input/simulink_2_plc_types.h, Logical/test_input/test_input.c, Logical/test_input/zero_crossing_types.h, Logical/test_input/extmode
